// SIMATIC S7-200 project (STEP 7-Micro/WIN), CPU 224 REL 01.22

ORGANIZATION_BLOCK MAIN:OB1
TITLE=PROGRAM COMMENTS
BEGIN
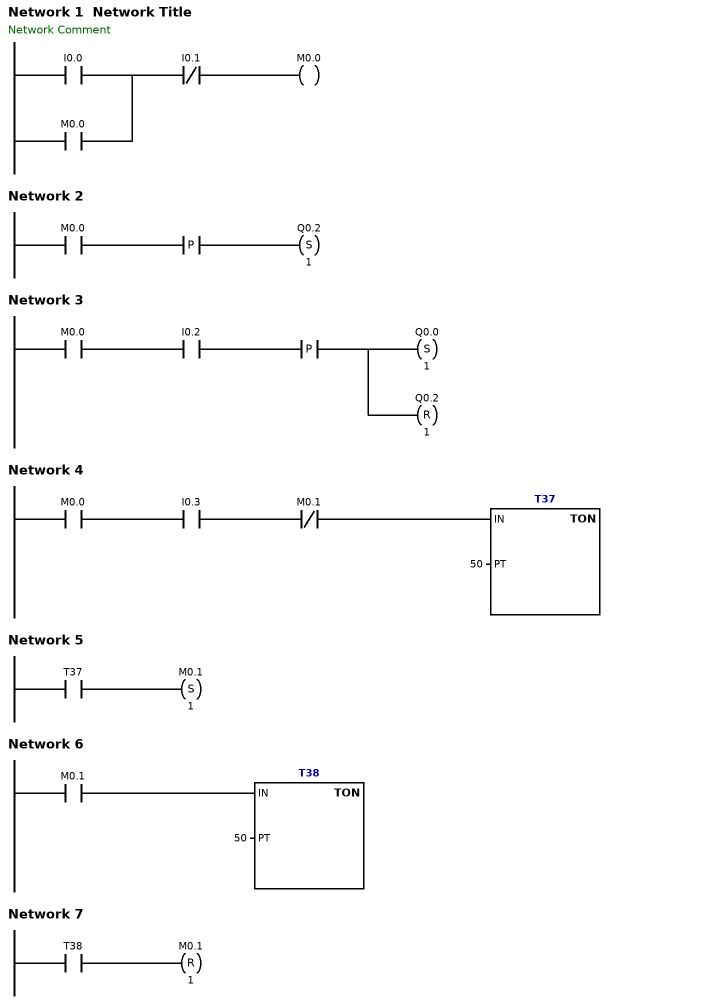
Network 1 // Network Title
// Network Comment
LD     I0.0
O      M0.0
AN     I0.1
=      M0.0
Network 2
LD     M0.0
EU
S      Q0.2, 1
Network 3
LD     M0.0
A      I0.2
EU
S      Q0.0, 1
R      Q0.2, 1
Network 4
LD     M0.0
A      I0.3
AN     M0.1
TON    T37, 50
Network 5
LD     T37
S      M0.1, 1
Network 6
LD     M0.1
TON    T38, 50
Network 7
LD     T38
R      M0.1, 1
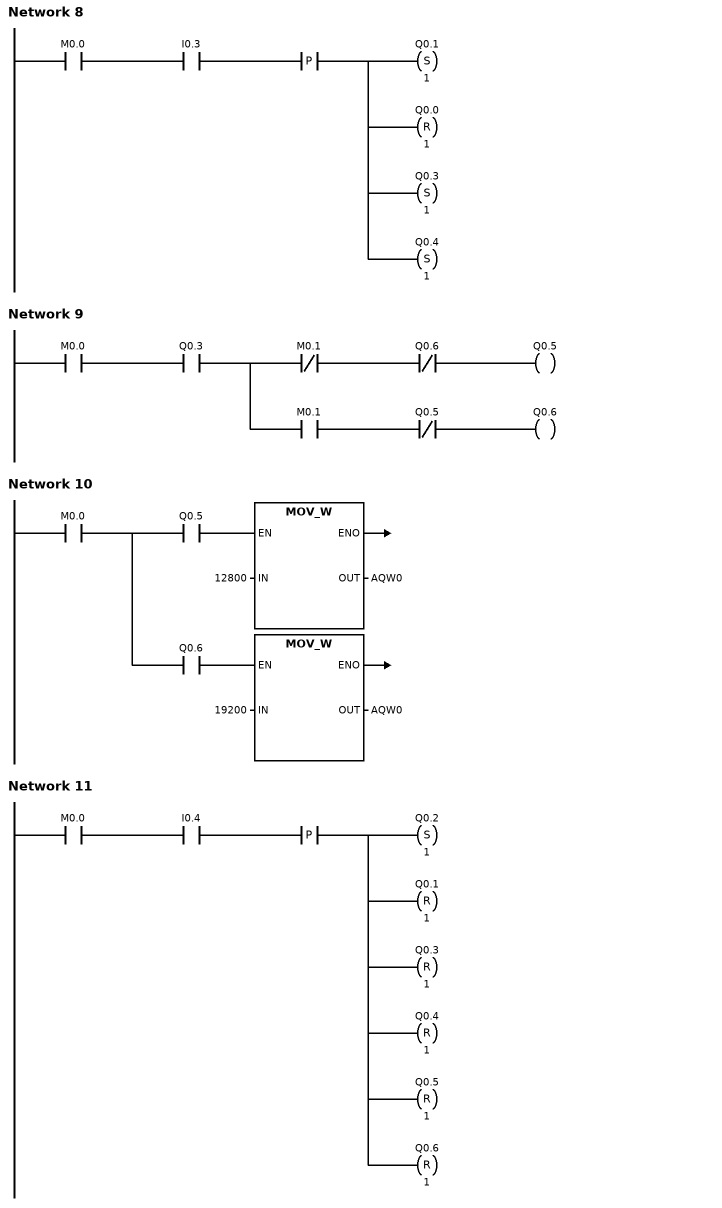
Network 8
LD     M0.0
A      I0.3
EU
S      Q0.1, 1
R      Q0.0, 1
S      Q0.3, 1
S      Q0.4, 1
Network 9
LD     M0.0
A      Q0.3
LPS
AN     M0.1
AN     Q0.6
=      Q0.5
LPP
A      M0.1
AN     Q0.5
=      Q0.6
Network 10
// (network saved uncompiled; LAD cells follow)
// row 0: c0 -| |- M0.0 v  c1 -| |- Q0.5  c2 [MOV_W EN:=power@row0, IN:=12800, ENO=>power, OUT=>AQW0]  c3 ->
// row 1: c0 ^v  c2 [box]
// row 2: c0 ^  c1 -| |- Q0.6  c2 [MOV_W EN:=power@row2, IN:=19200, ENO=>power, OUT=>AQW0]  c3 ->
// row 3: c2 [box]
Network 11
LD     M0.0
A      I0.4
EU
S      Q0.2, 1
R      Q0.1, 1
R      Q0.3, 1
R      Q0.4, 1
R      Q0.5, 1
R      Q0.6, 1
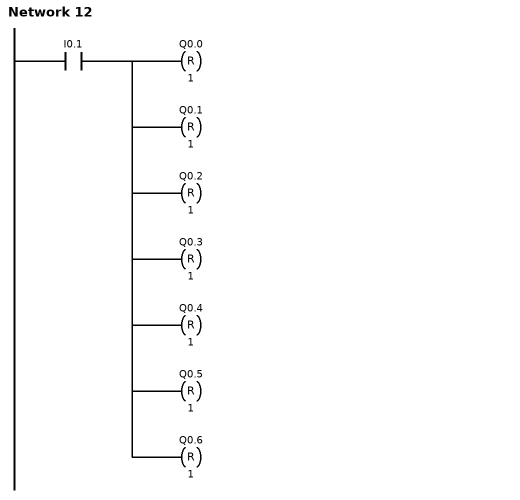
Network 12
LD     I0.1
R      Q0.0, 1
R      Q0.1, 1
R      Q0.2, 1
R      Q0.3, 1
R      Q0.4, 1
R      Q0.5, 1
R      Q0.6, 1
END_ORGANIZATION_BLOCK
